// TIA Portal V17 export
// export: Created 2025-06-26T06:49:34.4295215Z, ExportSetting WithDefaults, DisplayName Totally Integrated Automation Portal, DisplayVersion V17 Update 8, DisplayName TIA Portal Openness, DisplayVersion V17 Update 8, DisplayName TIA Portal Version Control Interface, DisplayVersion V17, DisplayName STEP 7 Professional, DisplayVersion V17 Update 8, DisplayName STEP 7 Safety, DisplayVersion V17 Update 6, DisplayName WinCC Advanced, DisplayVersion V17 Update 8
VAR_GLOBAL   // PLC tag table "RIO1"
   RIO1_Slot4_I AT %I634.0 : "stSM531_8AI";   //    {ExternalAccessible false, ExternalVisible false, ExternalWritable false}
   RIO1_Slot2_I AT %I600.0 : "stSM531_8AI";   //    {ExternalAccessible false, ExternalVisible false, ExternalWritable false}
   RIO1_Slot3_I AT %I617.0 : "stSM531_8AI";   //    {ExternalAccessible false, ExternalVisible false, ExternalWritable false}
   RIO1_Slot5_I AT %I651.0 : "stSM531_8AI";   //    {ExternalAccessible false, ExternalVisible false, ExternalWritable false}
   RIO1_Slot6_I AT %I668.0 : "stSM531_8AI";   //    {ExternalAccessible false, ExternalVisible false, ExternalWritable false}
   RIO1_Slot7_I AT %I685.0 : "stSM531_8AI";   //    {ExternalAccessible false, ExternalVisible false, ExternalWritable false}
   RIO1_Slot8_I AT %I702.0 : "stSM531_8AI";   //    {ExternalAccessible false, ExternalVisible false, ExternalWritable false}
   RIO1_Slot9_I AT %I719.0 : "stSM531_8AI";   //    {ExternalAccessible false, ExternalVisible false, ExternalWritable false}
   RIO1_Slot10_I AT %I736.0 : "stSM531_8AI";   //    {ExternalAccessible false, ExternalVisible false, ExternalWritable false}
   RIO1_Slot11_I AT %I753.0 : "stSM531_8AI";   //    {ExternalAccessible false, ExternalVisible false, ExternalWritable false}
   RIO1_Slot12_I AT %I770.0 : "stSM531_8AI";   //    {ExternalAccessible false, ExternalVisible false, ExternalWritable false}
   RIO1_Slot13_I AT %I787.0 : "stSM521_16DI";   //    {ExternalAccessible false, ExternalVisible false, ExternalWritable false}
   RIO1_Slot14_I AT %I789.0 : "stSM531_8AQ_I";   //    {ExternalAccessible false, ExternalVisible false, ExternalWritable false}
   RIO1_Slot15_I AT %I790.0 : "stSM531_8AQ_I";   //    {ExternalAccessible false, ExternalVisible false, ExternalWritable false}
   RIO1_Slot16_I AT %I791.0 : "stSM522_32DQ_I";   //    {ExternalAccessible false, ExternalVisible false, ExternalWritable false}
   RIO1_Slot14_Q AT %Q600.0 : "stSM531_8AQ";   //    {ExternalAccessible false, ExternalVisible false, ExternalWritable false}
   RIO1_Slot15_Q AT %Q616.0 : "stSM531_8AQ";   //    {ExternalAccessible false, ExternalVisible false, ExternalWritable false}
   RIO1_Slot16_Q AT %Q632.0 : "stSM522_32DQ_Q";   //    {ExternalAccessible false, ExternalVisible false, ExternalWritable false}
END_VAR
